ABB RobotStudio station: LogoTesla.rsstnx

Station LogoTesla (saved by RobotStudio 23.4.10609.1)
Controller IRB140_6_81
  mechanical unit ROB_1: IRB140_6_81_C_03, 6 joints, base frame (0, 0, 0) mm
Layout (positions relative to the parent item):
  - IRB140_6_81_C_03 [mechanism, from %ABB.RobotStudio.Models.IRB140%\IRB140_6_81_C_G_03.rslib] at (0, 0, 0) mm; joint values [0, 0, 0, 0, 0.5236, 0] (rad or m)
  - PenTool [part] at (506.29, 0, 679.5) mm, rotated rx 180 ry 60 rz 180 deg, size 50 x 102.1 x 106.1 mm
  - Marxador [mechanism] at (506.29, 0, 679.5) mm, rotated rx 180 ry 60 rz 180 deg
      TCP Marxador at (0, 35, -0.01) mm, rotated rx -90 ry 0 rz 0 deg
      links: Marcador
  - Base [part] at (500, 145, 0) mm, rotated rx 90 ry 0 rz -90 deg, size 288 x 191.6 x 383.2 mm
Attachment: Marxador is attached to IRB140_6_81_C_03 / Link6
Attachment: PenTool is attached to IRB140_6_81_C_03 / Link6
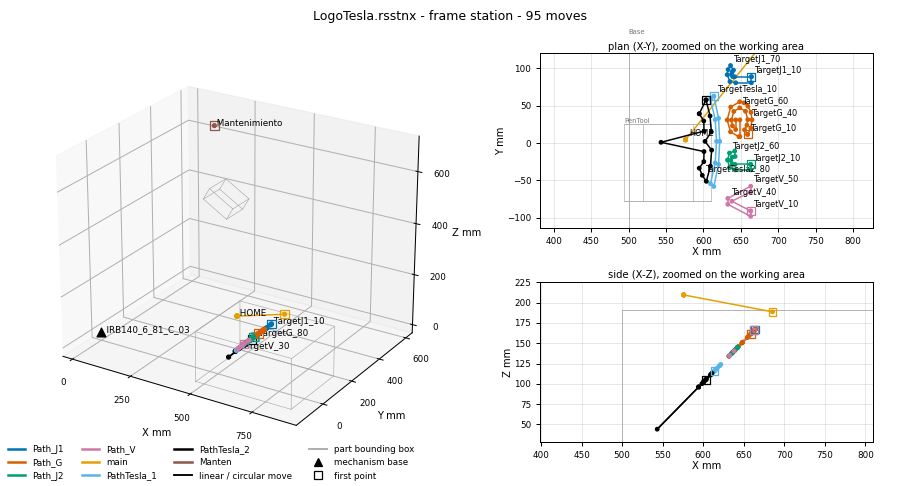
[picture p0: tool path of LogoTesla.rsstnx in frame station, 95 of 95 moves have a stored position in this frame; points joined in program order, loops and branches not executed]
Targets, tools, work objects and paths stored in the station, written as RAPID:
! task T_ROB1
MODULE Module1
  PERS tooldata Marxador:=[TRUE,[[0,-95.455,124.465],[0.923879533,0.382683432,0,0]],[1,[0,0,1],[1,0,0,0],0,0,0]];
  CONST robtarget TargetJ1_10:=[[664.045,88.658,166.933],[0.273445943,-0.652094561,0.652094561,-0.273445943],[0,0,0,0],[9E+09,9E+09,9E+09,9E+09,9E+09,9E+09]];
  CONST robtarget TargetJ1_20:=[[664.045,80.585,166.933],[0.273445943,-0.652094561,0.652094561,-0.273445943],[0,0,0,0],[9E+09,9E+09,9E+09,9E+09,9E+09,9E+09]];
  CONST robtarget TargetJ1_30:=[[643.116,80.585,145.635],[0.273445943,-0.652094561,0.652094561,-0.273445943],[0,0,0,0],[9E+09,9E+09,9E+09,9E+09,9E+09,9E+09]];
  CONST robtarget TargetJ1_40:=[[635.402,82.132,137.786],[0.273445943,-0.652094561,0.652094561,-0.273445943],[0,0,0,0],[9E+09,9E+09,9E+09,9E+09,9E+09,9E+09]];
  CONST robtarget TargetJ1_50:=[[631.71,91.361,134.029],[0.273445943,-0.652094561,0.652094561,-0.273445943],[0,0,0,0],[9E+09,9E+09,9E+09,9E+09,9E+09,9E+09]];
  CONST robtarget TargetJ1_60:=[[632.909,98.256,135.249],[0.273445943,-0.652094561,0.652094561,-0.273445943],[0,0,0,0],[9E+09,9E+09,9E+09,9E+09,9E+09,9E+09]];
  CONST robtarget TargetJ1_70:=[[636.175,103.651,138.573],[0.273445943,-0.652094561,0.652094561,-0.273445943],[0,0,0,0],[9E+09,9E+09,9E+09,9E+09,9E+09,9E+09]];
  CONST robtarget TargetJ1_80:=[[640.135,97.542,142.602],[0.273445943,-0.652094561,0.652094561,-0.273445943],[0,0,0,0],[9E+09,9E+09,9E+09,9E+09,9E+09,9E+09]];
  CONST robtarget TargetJ1_90:=[[638.277,94.845,140.711],[0.273445943,-0.652094561,0.652094561,-0.273445943],[0,0,0,0],[9E+09,9E+09,9E+09,9E+09,9E+09,9E+09]];
  CONST robtarget TargetJ1_100:=[[637.369,91.352,139.787],[0.273445943,-0.652094561,0.652094561,-0.273445943],[0,0,0,0],[9E+09,9E+09,9E+09,9E+09,9E+09,9E+09]];
  CONST robtarget TargetJ1_110:=[[639.114,88.909,141.564],[0.273445943,-0.652094561,0.652094561,-0.273445943],[0,0,0,0],[9E+09,9E+09,9E+09,9E+09,9E+09,9E+09]];
  CONST robtarget TargetJ1_120:=[[641.802,88.658,144.299],[0.273445943,-0.652094561,0.652094561,-0.273445943],[0,0,0,0],[9E+09,9E+09,9E+09,9E+09,9E+09,9E+09]];
  CONST robtarget TargetG_10:=[[659.03,11.683,161.83],[0.273445943,-0.652094561,0.652094561,-0.273445943],[0,0,0,0],[9E+09,9E+09,9E+09,9E+09,9E+09,9E+09]];
  CONST robtarget TargetG_20:=[[654.932,17.792,157.66],[0.273445943,-0.652094561,0.652094561,-0.273445943],[0,0,0,0],[9E+09,9E+09,9E+09,9E+09,9E+09,9E+09]];
  CONST robtarget TargetG_30:=[[658.076,23.913,160.859],[0.273445943,-0.652094561,0.652094561,-0.273445943],[0,0,0,0],[9E+09,9E+09,9E+09,9E+09,9E+09,9E+09]];
  CONST robtarget TargetG_40:=[[659.195,31.316,161.998],[0.273445943,-0.652094561,0.652094561,-0.273445943],[0,0,0,0],[9E+09,9E+09,9E+09,9E+09,9E+09,9E+09]];
  CONST robtarget TargetG_50:=[[656.148,42.472,158.897],[0.273445943,-0.652094561,0.652094561,-0.273445943],[0,0,0,0],[9E+09,9E+09,9E+09,9E+09,9E+09,9E+09]];
  CONST robtarget TargetG_60:=[[648.446,47.138,151.06],[0.273445943,-0.652094561,0.652094561,-0.273445943],[0,0,0,0],[9E+09,9E+09,9E+09,9E+09,9E+09,9E+09]];
  CONST robtarget TargetG_70:=[[640.497,42.263,142.971],[0.273445943,-0.652094561,0.652094561,-0.273445943],[0,0,0,0],[9E+09,9E+09,9E+09,9E+09,9E+09,9E+09]];
  CONST robtarget TargetG_80:=[[637.369,30.704,139.787],[0.273445943,-0.652094561,0.652094561,-0.273445943],[0,0,0,0],[9E+09,9E+09,9E+09,9E+09,9E+09,9E+09]];
  CONST robtarget TargetG_90:=[[638.749,23.067,141.192],[0.273445943,-0.652094561,0.652094561,-0.273445943],[0,0,0,0],[9E+09,9E+09,9E+09,9E+09,9E+09,9E+09]];
  CONST robtarget TargetG_100:=[[643.027,18.08,145.546],[0.273445943,-0.652094561,0.652094561,-0.273445943],[0,0,0,0],[9E+09,9E+09,9E+09,9E+09,9E+09,9E+09]];
  CONST robtarget TargetG_110:=[[643.027,30.992,145.546],[0.273445943,-0.652094561,0.652094561,-0.273445943],[0,0,0,0],[9E+09,9E+09,9E+09,9E+09,9E+09,9E+09]];
  CONST robtarget TargetG_120:=[[648.686,30.992,151.304],[0.273445943,-0.652094561,0.652094561,-0.273445943],[0,0,0,0],[9E+09,9E+09,9E+09,9E+09,9E+09,9E+09]];
  CONST robtarget TargetG_130:=[[648.686,8.566,151.304],[0.273445943,-0.652094561,0.652094561,-0.273445943],[0,0,0,0],[9E+09,9E+09,9E+09,9E+09,9E+09,9E+09]];
  CONST robtarget TargetG_140:=[[647.341,8.503,149.935],[0.273445943,-0.652094561,0.652094561,-0.273445943],[0,0,0,0],[9E+09,9E+09,9E+09,9E+09,9E+09,9E+09]];
  CONST robtarget TargetG_150:=[[636.165,14.971,138.563],[0.273445943,-0.652094561,0.652094561,-0.273445943],[0,0,0,0],[9E+09,9E+09,9E+09,9E+09,9E+09,9E+09]];
  CONST robtarget TargetG_160:=[[631.71,30.866,134.029],[0.273445943,-0.652094561,0.652094561,-0.273445943],[0,0,0,0],[9E+09,9E+09,9E+09,9E+09,9E+09,9E+09]];
  CONST robtarget TargetG_170:=[[636.388,48.19,138.789],[0.273445943,-0.652094561,0.652094561,-0.273445943],[0,0,0,0],[9E+09,9E+09,9E+09,9E+09,9E+09,9E+09]];
  CONST robtarget TargetG_180:=[[648.439,55.212,151.053],[0.273445943,-0.652094561,0.652094561,-0.273445943],[0,0,0,0],[9E+09,9E+09,9E+09,9E+09,9E+09,9E+09]];
  CONST robtarget TargetG_190:=[[654.284,53.743,157.001],[0.273445943,-0.652094561,0.652094561,-0.273445943],[0,0,0,0],[9E+09,9E+09,9E+09,9E+09,9E+09,9E+09]];
  CONST robtarget TargetG_200:=[[659.34,49.31,162.145],[0.273445943,-0.652094561,0.652094561,-0.273445943],[0,0,0,0],[9E+09,9E+09,9E+09,9E+09,9E+09,9E+09]];
  CONST robtarget TargetG_210:=[[663.525,41.09,166.405],[0.273445943,-0.652094561,0.652094561,-0.273445943],[0,0,0,0],[9E+09,9E+09,9E+09,9E+09,9E+09,9E+09]];
  CONST robtarget TargetG_220:=[[664.853,31.091,167.756],[0.273445943,-0.652094561,0.652094561,-0.273445943],[0,0,0,0],[9E+09,9E+09,9E+09,9E+09,9E+09,9E+09]];
  CONST robtarget TargetG_230:=[[663.363,20.117,166.239],[0.273445943,-0.652094561,0.652094561,-0.273445943],[0,0,0,0],[9E+09,9E+09,9E+09,9E+09,9E+09,9E+09]];
  CONST robtarget TargetJ2_10:=[[663.121,-28.591,165.993],[0.273445943,-0.652094561,0.652094561,-0.273445943],[-1,0,-2,0],[9E+09,9E+09,9E+09,9E+09,9E+09,9E+09]];
  CONST robtarget TargetJ2_20:=[[663.121,-35.868,165.993],[0.273445943,-0.652094561,0.652094561,-0.273445943],[0,0,0,0],[9E+09,9E+09,9E+09,9E+09,9E+09,9E+09]];
  CONST robtarget TargetJ2_30:=[[642.529,-35.868,145.039],[0.273445943,-0.652094561,0.652094561,-0.273445943],[0,0,0,0],[9E+09,9E+09,9E+09,9E+09,9E+09,9E+09]];
  CONST robtarget TargetJ2_40:=[[634.983,-32.958,137.36],[0.273445943,-0.652094561,0.652094561,-0.273445943],[0,0,0,0],[9E+09,9E+09,9E+09,9E+09,9E+09,9E+09]];
  CONST robtarget TargetJ2_50:=[[632.126,-22.748,134.452],[0.273445943,-0.652094561,0.652094561,-0.273445943],[0,0,0,0],[9E+09,9E+09,9E+09,9E+09,9E+09,9E+09]];
  CONST robtarget TargetJ2_60:=[[634.788,-13.325,137.162],[0.273445943,-0.652094561,0.652094561,-0.273445943],[0,0,0,0],[9E+09,9E+09,9E+09,9E+09,9E+09,9E+09]];
  CONST robtarget TargetJ2_70:=[[641.794,-10.678,144.29],[0.273445943,-0.652094561,0.652094561,-0.273445943],[0,0,0,0],[9E+09,9E+09,9E+09,9E+09,9E+09,9E+09]];
  CONST robtarget TargetJ2_80:=[[642.327,-17.929,144.833],[0.273445943,-0.652094561,0.652094561,-0.273445943],[0,0,0,0],[9E+09,9E+09,9E+09,9E+09,9E+09,9E+09]];
  CONST robtarget TargetJ2_90:=[[638.505,-18.749,140.943],[0.273445943,-0.652094561,0.652094561,-0.273445943],[0,0,0,0],[9E+09,9E+09,9E+09,9E+09,9E+09,9E+09]];
  CONST robtarget TargetJ2_100:=[[636.442,-23.037,138.844],[0.273445943,-0.652094561,0.652094561,-0.273445943],[0,0,0,0],[9E+09,9E+09,9E+09,9E+09,9E+09,9E+09]];
  CONST robtarget TargetJ2_110:=[[638.302,-27.82,140.738],[0.273445943,-0.652094561,0.652094561,-0.273445943],[0,0,0,0],[9E+09,9E+09,9E+09,9E+09,9E+09,9E+09]];
  CONST robtarget TargetJ2_120:=[[642.315,-28.591,144.82],[0.273445943,-0.652094561,0.652094561,-0.273445943],[0,0,0,0],[9E+09,9E+09,9E+09,9E+09,9E+09,9E+09]];
  CONST robtarget TargetV_10:=[[663.121,-90.794,165.993],[0.273445943,-0.652094561,0.652094561,-0.273445943],[-1,0,-2,0],[9E+09,9E+09,9E+09,9E+09,9E+09,9E+09]];
  CONST robtarget TargetV_20:=[[663.121,-98.001,165.993],[0.273445943,-0.652094561,0.652094561,-0.273445943],[0,0,0,0],[9E+09,9E+09,9E+09,9E+09,9E+09,9E+09]];
  CONST robtarget TargetV_30:=[[632.518,-81.864,134.852],[0.273445943,-0.652094561,0.652094561,-0.273445943],[0,0,0,0],[9E+09,9E+09,9E+09,9E+09,9E+09,9E+09]];
  CONST robtarget TargetV_40:=[[632.518,-73.958,134.852],[0.273445943,-0.652094561,0.652094561,-0.273445943],[0,0,0,0],[9E+09,9E+09,9E+09,9E+09,9E+09,9E+09]];
  CONST robtarget TargetV_50:=[[663.121,-57.698,165.993],[0.273445943,-0.652094561,0.652094561,-0.273445943],[0,0,0,0],[9E+09,9E+09,9E+09,9E+09,9E+09,9E+09]];
  CONST robtarget TargetV_60:=[[663.121,-65.238,165.993],[0.273445943,-0.652094561,0.652094561,-0.273445943],[0,0,0,0],[9E+09,9E+09,9E+09,9E+09,9E+09,9E+09]];
  CONST robtarget TargetV_70:=[[637.983,-77.783,140.413],[0.273445943,-0.652094561,0.652094561,-0.273445943],[0,0,0,0],[9E+09,9E+09,9E+09,9E+09,9E+09,9E+09]];
  CONST robtarget HOME:=[[575.945734827,4.319172051,209.541129224],[0.273941946,-0.670576408,0.638463051,-0.260092335],[-1,0,-2,0],[9E+09,9E+09,9E+09,9E+09,9E+09,9E+09]];
  CONST robtarget TargetTesla_10:=[[613.873,62.613,115.878],[0.273445943,-0.652094561,0.652094561,-0.273445943],[0,0,0,0],[9E+09,9E+09,9E+09,9E+09,9E+09,9E+09]];
  CONST robtarget TargetTesla_20:=[[620.169,33.102,122.285],[0.273445943,-0.652094561,0.652094561,-0.273445943],[0,0,0,0],[9E+09,9E+09,9E+09,9E+09,9E+09,9E+09]];
  CONST robtarget TargetTesla_30:=[[621.7,2.278,123.843],[0.273445943,-0.652094561,0.652094561,-0.273445943],[0,0,0,0],[9E+09,9E+09,9E+09,9E+09,9E+09,9E+09]];
  CONST robtarget TargetTesla_40:=[[620.169,-28.545,122.285],[0.273445943,-0.652094561,0.652094561,-0.273445943],[0,0,0,0],[9E+09,9E+09,9E+09,9E+09,9E+09,9E+09]];
  CONST robtarget TargetTesla_50:=[[613.873,-58.056,115.878],[0.273445943,-0.652094561,0.652094561,-0.273445943],[0,0,0,0],[9E+09,9E+09,9E+09,9E+09,9E+09,9E+09]];
  CONST robtarget TargetTesla_60:=[[609.365,-54.276,111.291],[0.273445943,-0.652094561,0.652094561,-0.273445943],[0,0,0,0],[9E+09,9E+09,9E+09,9E+09,9E+09,9E+09]];
  CONST robtarget TargetTesla_70:=[[615.652,-26.644,117.688],[0.273445943,-0.652094561,0.652094561,-0.273445943],[0,0,0,0],[9E+09,9E+09,9E+09,9E+09,9E+09,9E+09]];
  CONST robtarget TargetTesla_80:=[[617.466,2.278,119.535],[0.273445943,-0.652094561,0.652094561,-0.273445943],[0,0,0,0],[9E+09,9E+09,9E+09,9E+09,9E+09,9E+09]];
  CONST robtarget TargetTesla_90:=[[615.652,31.201,117.688],[0.273445943,-0.652094561,0.652094561,-0.273445943],[0,0,0,0],[9E+09,9E+09,9E+09,9E+09,9E+09,9E+09]];
  CONST robtarget TargetTesla_100:=[[609.365,58.833,111.291],[0.273445943,-0.652094561,0.652094561,-0.273445943],[0,0,0,0],[9E+09,9E+09,9E+09,9E+09,9E+09,9E+09]];
  CONST robtarget TargetTesla2_10:=[[603.376,57.695,105.196],[0.273445943,-0.652094561,0.652094561,-0.273445943],[0,0,0,0],[9E+09,9E+09,9E+09,9E+09,9E+09,9E+09]];
  CONST robtarget TargetTesla2_20:=[[608.815,36.23,110.731],[0.273445943,-0.652094561,0.652094561,-0.273445943],[0,0,0,0],[9E+09,9E+09,9E+09,9E+09,9E+09,9E+09]];
  CONST robtarget TargetTesla2_30:=[[610.48,14.932,112.425],[0.273445943,-0.652094561,0.652094561,-0.273445943],[0,0,0,0],[9E+09,9E+09,9E+09,9E+09,9E+09,9E+09]];
  CONST robtarget TargetTesla2_40:=[[602.075,2.278,103.872],[0.273445943,-0.652094561,0.652094561,-0.273445943],[0,0,0,0],[9E+09,9E+09,9E+09,9E+09,9E+09,9E+09]];
  CONST robtarget TargetTesla2_50:=[[610.928,-9.422,112.881],[0.273445943,-0.652094561,0.652094561,-0.273445943],[0,0,0,0],[9E+09,9E+09,9E+09,9E+09,9E+09,9E+09]];
  CONST robtarget TargetTesla2_60:=[[609.268,-30.956,111.192],[0.273445943,-0.652094561,0.652094561,-0.273445943],[0,0,0,0],[9E+09,9E+09,9E+09,9E+09,9E+09,9E+09]];
  CONST robtarget TargetTesla2_70:=[[603.802,-51.159,105.63],[0.273445943,-0.652094561,0.652094561,-0.273445943],[0,0,0,0],[9E+09,9E+09,9E+09,9E+09,9E+09,9E+09]];
  CONST robtarget TargetTesla2_80:=[[598.396,-43.097,100.129],[0.273445943,-0.652094561,0.652094561,-0.273445943],[0,0,0,0],[9E+09,9E+09,9E+09,9E+09,9E+09,9E+09]];
  CONST robtarget TargetTesla2_90:=[[594.348,-33.576,96.009],[0.273445943,-0.652094561,0.652094561,-0.273445943],[0,0,0,0],[9E+09,9E+09,9E+09,9E+09,9E+09,9E+09]];
  CONST robtarget TargetTesla2_100:=[[600.439,-24.871,102.207],[0.273445943,-0.652094561,0.652094561,-0.273445943],[0,0,0,0],[9E+09,9E+09,9E+09,9E+09,9E+09,9E+09]];
  CONST robtarget TargetTesla2_110:=[[600.71,-11.382,102.483],[0.273445943,-0.652094561,0.652094561,-0.273445943],[0,0,0,0],[9E+09,9E+09,9E+09,9E+09,9E+09,9E+09]];
  CONST robtarget TargetTesla2_120:=[[543.238,1,43.999],[0.273445943,-0.652094561,0.652094561,-0.273445943],[0,0,0,0],[9E+09,9E+09,9E+09,9E+09,9E+09,9E+09]];
  CONST robtarget TargetTesla2_130:=[[600.71,15.939,102.483],[0.273445943,-0.652094561,0.652094561,-0.273445943],[0,0,0,0],[9E+09,9E+09,9E+09,9E+09,9E+09,9E+09]];
  CONST robtarget TargetTesla2_140:=[[600.418,29.549,102.186],[0.273445943,-0.652094561,0.652094561,-0.273445943],[0,0,0,0],[9E+09,9E+09,9E+09,9E+09,9E+09,9E+09]];
  CONST robtarget TargetTesla2_150:=[[594.369,39.16,96.031],[0.273445943,-0.652094561,0.652094561,-0.273445943],[0,0,0,0],[9E+09,9E+09,9E+09,9E+09,9E+09,9E+09]];
  CONST robtarget Posicion_Inicial:=[[685.464,141,188.73],[0.273445943,-0.652094561,0.652094561,-0.273445943],[0,-1,-1,0],[9E+09,9E+09,9E+09,9E+09,9E+09,9E+09]];
  CONST robtarget Mantenimiento:=[[95.455040021,614.081531206,617.267467743],[0.560985581,-0.430459309,0.70105737,0.092295858],[1,-1,0,0],[9E+09,9E+09,9E+09,9E+09,9E+09,9E+09]];
  PROC Path_J1()
    MoveL TargetJ1_10,v100,z100,Marxador\WObj:=wobj0;
    MoveL TargetJ1_20,v100,z100,Marxador\WObj:=wobj0;
    MoveL TargetJ1_30,v100,z100,Marxador\WObj:=wobj0;
    MoveL TargetJ1_40,v100,z10,Marxador\WObj:=wobj0;
    MoveL TargetJ1_50,v100,z10,Marxador\WObj:=wobj0;
    MoveL TargetJ1_60,v100,z100,Marxador\WObj:=wobj0;
    MoveL TargetJ1_70,v100,z100,Marxador\WObj:=wobj0;
    MoveL TargetJ1_80,v100,z100,Marxador\WObj:=wobj0;
    MoveL TargetJ1_90,v100,z100,Marxador\WObj:=wobj0;
    MoveL TargetJ1_100,v100,z100,Marxador\WObj:=wobj0;
    MoveL TargetJ1_110,v100,z100,Marxador\WObj:=wobj0;
    MoveL TargetJ1_120,v100,z100,Marxador\WObj:=wobj0;
    MoveL TargetJ1_10,v50,z0,Marxador\WObj:=wobj0;
  ENDPROC
  PROC Path_G()
    MoveL TargetG_10,v100,z100,Marxador\WObj:=wobj0;
    MoveL TargetG_20,v100,z100,Marxador\WObj:=wobj0;
    MoveL TargetG_30,v100,z100,Marxador\WObj:=wobj0;
    MoveL TargetG_40,v100,z100,Marxador\WObj:=wobj0;
    MoveL TargetG_50,v100,z100,Marxador\WObj:=wobj0;
    MoveL TargetG_60,v100,z100,Marxador\WObj:=wobj0;
    MoveL TargetG_70,v100,z100,Marxador\WObj:=wobj0;
    MoveL TargetG_80,v100,z100,Marxador\WObj:=wobj0;
    MoveL TargetG_90,v100,z100,Marxador\WObj:=wobj0;
    MoveL TargetG_100,v100,z100,Marxador\WObj:=wobj0;
    MoveL TargetG_110,v100,z100,Marxador\WObj:=wobj0;
    MoveL TargetG_120,v100,z100,Marxador\WObj:=wobj0;
    MoveL TargetG_130,v100,z100,Marxador\WObj:=wobj0;
    MoveL TargetG_140,v100,z100,Marxador\WObj:=wobj0;
    MoveL TargetG_150,v100,z100,Marxador\WObj:=wobj0;
    MoveL TargetG_160,v100,z100,Marxador\WObj:=wobj0;
    MoveL TargetG_170,v100,z100,Marxador\WObj:=wobj0;
    MoveL TargetG_180,v100,z100,Marxador\WObj:=wobj0;
    MoveL TargetG_190,v100,z100,Marxador\WObj:=wobj0;
    MoveL TargetG_200,v100,z100,Marxador\WObj:=wobj0;
    MoveL TargetG_210,v100,z100,Marxador\WObj:=wobj0;
    MoveL TargetG_220,v100,z100,Marxador\WObj:=wobj0;
    MoveL TargetG_230,v100,z100,Marxador\WObj:=wobj0;
    MoveL TargetG_10,v50,z0,Marxador\WObj:=wobj0;
  ENDPROC
  PROC Path_J2()
    MoveL TargetJ2_10,v100,z100,Marxador\WObj:=wobj0;
    MoveL TargetJ2_20,v100,z100,Marxador\WObj:=wobj0;
    MoveL TargetJ2_30,v100,z100,Marxador\WObj:=wobj0;
    MoveL TargetJ2_40,v100,z100,Marxador\WObj:=wobj0;
    MoveL TargetJ2_50,v100,z100,Marxador\WObj:=wobj0;
    MoveL TargetJ2_60,v100,z100,Marxador\WObj:=wobj0;
    MoveL TargetJ2_70,v100,z100,Marxador\WObj:=wobj0;
    MoveL TargetJ2_80,v100,z100,Marxador\WObj:=wobj0;
    MoveL TargetJ2_90,v100,z100,Marxador\WObj:=wobj0;
    MoveL TargetJ2_100,v100,z100,Marxador\WObj:=wobj0;
    MoveL TargetJ2_110,v100,z100,Marxador\WObj:=wobj0;
    MoveL TargetJ2_120,v100,z100,Marxador\WObj:=wobj0;
    MoveL TargetJ2_10,v50,z0,Marxador\WObj:=wobj0;
  ENDPROC
  PROC Path_V()
    MoveL TargetV_10,v100,z100,Marxador\WObj:=wobj0;
    MoveL TargetV_20,v100,z100,Marxador\WObj:=wobj0;
    MoveL TargetV_30,v100,z100,Marxador\WObj:=wobj0;
    MoveL TargetV_40,v100,z100,Marxador\WObj:=wobj0;
    MoveL TargetV_50,v100,z100,Marxador\WObj:=wobj0;
    MoveL TargetV_60,v100,z100,Marxador\WObj:=wobj0;
    MoveL TargetV_70,v100,z100,Marxador\WObj:=wobj0;
    MoveL TargetV_10,v50,z0,Marxador\WObj:=wobj0;
  ENDPROC
  PROC main()
    Reset L_OutDO_Maintance;
    Reset L_OutDO_Origin;
    Reset L_OutDO_Start;
    WaitDI L_IntDI_Maintance,1;
    Set L_OutDO_Maintance;
    Manten;
    WaitDI L_IntDI_Origin,1;
    Reset L_OutDO_Maintance;
    Set L_OutDO_Origin;
    MoveJ Posicion_Inicial,v100,z100,Marxador\WObj:=wobj0;
    WaitDI L_IntDI_Start,1;
    Reset L_OutDO_Origin;
    Set L_OutDO_Start;
    MoveL HOME,v100,z100,Marxador\WObj:=wobj0;
    Path_J1;
    MoveL HOME,v100,z100,Marxador\WObj:=wobj0;
    Path_G;
    MoveL HOME,v100,z100,Marxador\WObj:=wobj0;
    Path_J2;
    MoveL HOME,v100,z100,Marxador\WObj:=wobj0;
    Path_V;
    MoveL HOME,v100,z100,Marxador\WObj:=wobj0;
    PathTesla_1;
    MoveL HOME,v100,z100,Marxador\WObj:=wobj0;
    PathTesla_2;
    MoveL HOME,v100,z100,Marxador\WObj:=wobj0;
    Reset L_OutDO_Start;
  ENDPROC
  PROC PathTesla_1()
    MoveL TargetTesla_10,v100,z100,Marxador\WObj:=wobj0;
    MoveL TargetTesla_20,v100,z100,Marxador\WObj:=wobj0;
    MoveL TargetTesla_30,v100,z100,Marxador\WObj:=wobj0;
    MoveL TargetTesla_40,v100,z100,Marxador\WObj:=wobj0;
    MoveL TargetTesla_50,v100,z100,Marxador\WObj:=wobj0;
    MoveL TargetTesla_60,v100,z100,Marxador\WObj:=wobj0;
    MoveL TargetTesla_70,v100,z100,Marxador\WObj:=wobj0;
    MoveL TargetTesla_80,v100,z100,Marxador\WObj:=wobj0;
    MoveL TargetTesla_90,v100,z100,Marxador\WObj:=wobj0;
    MoveL TargetTesla_100,v100,z100,Marxador\WObj:=wobj0;
    MoveL TargetTesla_10,v50,z100,Marxador\WObj:=wobj0;
  ENDPROC
  PROC PathTesla_2()
    MoveL TargetTesla2_10,v100,z100,Marxador\WObj:=wobj0;
    MoveL TargetTesla2_20,v100,z100,Marxador\WObj:=wobj0;
    MoveL TargetTesla2_30,v100,z100,Marxador\WObj:=wobj0;
    MoveL TargetTesla2_40,v100,z100,Marxador\WObj:=wobj0;
    MoveL TargetTesla2_50,v100,z100,Marxador\WObj:=wobj0;
    MoveL TargetTesla2_60,v100,z100,Marxador\WObj:=wobj0;
    MoveL TargetTesla2_70,v100,z100,Marxador\WObj:=wobj0;
    MoveL TargetTesla2_80,v100,z100,Marxador\WObj:=wobj0;
    MoveL TargetTesla2_90,v100,z10,Marxador\WObj:=wobj0;
    MoveL TargetTesla2_100,v100,z100,Marxador\WObj:=wobj0;
    MoveL TargetTesla2_110,v100,z100,Marxador\WObj:=wobj0;
    MoveL TargetTesla2_120,v50,z0,Marxador\WObj:=wobj0;
    MoveL TargetTesla2_130,v100,z100,Marxador\WObj:=wobj0;
    MoveL TargetTesla2_140,v100,z100,Marxador\WObj:=wobj0;
    MoveL TargetTesla2_150,v100,z100,Marxador\WObj:=wobj0;
    MoveL TargetTesla2_150,v100,z100,Marxador\WObj:=wobj0;
    MoveL TargetTesla2_10,v100,z100,Marxador\WObj:=wobj0;
  ENDPROC
  PROC Manten()
    MoveJ Mantenimiento,v1000,z100,Marxador\WObj:=wobj0;
  ENDPROC
ENDMODULE

